(* IEC 61131-3 sources: tfc-hmi/packages/tfc_mcp_server/test/compiler/fixtures/common, 6 files *)

(* ---- type_declarations.st ---- *)
TYPE MotorState :
(
  Idle := 0,
  Starting := 1,
  Running := 2,
  Stopping := 3,
  Faulted := 4
);
END_TYPE

TYPE ST_MotorData :
STRUCT
  speed : REAL;
  current : REAL;
  temperature : REAL;
  state : MotorState;
  faultCode : DINT;
  name : STRING[32];
END_STRUCT
END_TYPE

TYPE AliasType : REAL;
END_TYPE

(* ---- function_example.st ---- *)
FUNCTION FC_Clamp : REAL
VAR_INPUT
  value : REAL;
  minVal : REAL;
  maxVal : REAL;
END_VAR
  IF value < minVal THEN
    FC_Clamp := minVal;
  ELSIF value > maxVal THEN
    FC_Clamp := maxVal;
  ELSE
    FC_Clamp := value;
  END_IF;
END_FUNCTION

(* ---- var_blocks.st ---- *)
FUNCTION_BLOCK FB_VarTest
VAR_INPUT
  enable : BOOL;
  setpoint : REAL;
  name : STRING[80];
END_VAR
VAR_OUTPUT
  done : BOOL;
  value : REAL;
END_VAR
VAR_IN_OUT
  counter : INT;
END_VAR
VAR
  internalState : INT;
  timer : INT;
END_VAR
VAR RETAIN
  retainedCount : DINT;
END_VAR
VAR CONSTANT
  MAX_VALUE : REAL := 100.0;
  MIN_VALUE : REAL := 0.0;
END_VAR
  IF enable THEN
    value := setpoint;
    done := TRUE;
  END_IF;
END_FUNCTION_BLOCK

(* ---- all_statements.st ---- *)
PROGRAM StatementTests
VAR
  i, j, state : INT;
  running : BOOL;
  speed, temp : REAL;
END_VAR
  // Simple assignment
  i := 42;

  // IF statement
  IF running THEN
    speed := 100.0;
  END_IF;

  // IF-ELSIF-ELSE
  IF temp > 80.0 THEN
    speed := 0.0;
  ELSIF temp > 60.0 THEN
    speed := 50.0;
  ELSIF temp > 40.0 THEN
    speed := 75.0;
  ELSE
    speed := 100.0;
  END_IF;

  // CASE statement
  CASE state OF
    0: speed := 0.0;
    1: speed := 50.0;
    2, 3: speed := 75.0;
    4..10: speed := 100.0;
  ELSE
    speed := 0.0;
  END_CASE;

  // FOR loop
  FOR i := 0 TO 9 DO
    j := j + i;
  END_FOR;

  // FOR with BY
  FOR i := 10 TO 0 BY -1 DO
    j := j + i;
  END_FOR;

  // WHILE loop
  WHILE running DO
    i := i + 1;
    IF i > 100 THEN
      running := FALSE;
    END_IF;
  END_WHILE;

  // REPEAT loop
  REPEAT
    i := i - 1;
  UNTIL i <= 0
  END_REPEAT;

  // EXIT
  FOR i := 0 TO 100 DO
    IF i = 50 THEN
      EXIT;
    END_IF;
  END_FOR;

  // RETURN
  RETURN;
END_PROGRAM

(* ---- expressions.st ---- *)
PROGRAM ExpressionTests
VAR
  a, b, c : INT;
  x, y : REAL;
  flag1, flag2, flag3 : BOOL;
  str1 : STRING[80];
  arr : ARRAY[1..10] OF INT;
END_VAR
  // Arithmetic
  a := 1 + 2;
  a := b - c;
  a := b * c;
  a := b / c;
  a := b MOD c;
  x := -y;

  // Comparison
  flag1 := a = b;
  flag1 := a <> b;
  flag1 := a < b;
  flag1 := a > b;
  flag1 := a <= b;
  flag1 := a >= b;

  // Boolean
  flag1 := flag2 AND flag3;
  flag1 := flag2 OR flag3;
  flag1 := flag2 XOR flag3;
  flag1 := NOT flag2;

  // Parenthesized
  a := (b + c) * 2;

  // Array access
  a := arr[1];
  arr[b + 1] := c;

  // Typed literals
  a := INT#42;
  x := REAL#3.14;

  // Time literal
  // (comment out for now - just have the file ready)

  // Nested expressions with precedence
  x := 1.0 + 2.0 * 3.0;
  flag1 := (a > 0) AND (b < 10) OR (c = 5);
END_PROGRAM

(* ---- fb_call_patterns.st ---- *)
PROGRAM FbCallTest
VAR
  timer1 : TON;
  motor : FB_Motor;
  result : REAL;
  elapsed : BOOL;
  capturedOutput : REAL;
END_VAR
  // Simple FB call
  timer1(IN := TRUE, PT := T#5s);
  elapsed := timer1.Q;

  // FB call with output capture
  motor(bStart := TRUE, rSetSpeed := 75.0, rActSpeed => capturedOutput);

  // Function call (positional)
  result := ABS(-42.0);

  // Function call (named)
  result := LIMIT(MN := 0.0, IN := result, MX := 100.0);

  // Chained member access
  result := motor.rActSpeed;
END_PROGRAM
